FUNCTION_BLOCK ExampleDomain_ExampleState EXTENDS _ExampleDomain_State

END_FUNCTION_BLOCK

(* stored: Version 1.1.0.1
   POU ExampleDomain_ExampleState: Id {3075723a-c4bd-49b6-8676-8704fb23a14f}, SpecialFunc None *)
